FUNCTION_BLOCK FB_Syntax_Derived EXTENDS FB_Syntax_AbstractBase IMPLEMENTS I_Syntax_Extended
VAR
    _sStatus  : STRING := 'IDLE';
    _nCounter : DINT;
END_VAR

_nCounter := _nCounter + 1;

METHOD M_Execute : BOOL
VAR_INPUT
    nCommand : DINT;
END_VAR
CASE nCommand OF
    1:
        _sStatus := 'RUNNING';
    2:
        _sStatus := 'PAUSED';
ELSE
    _sStatus := 'UNKNOWN';
END_CASE
M_Execute := TRUE;
END_METHOD

METHOD M_GetValue : INT
M_GetValue := TO_INT(_nCounter);
END_METHOD

METHOD M_Reset : BOOL
_nCounter := 0;
_bReady   := TRUE;
_sStatus  := 'RESET';
M_Reset   := TRUE;
END_METHOD

PROPERTY P_ExtendedStatus : INT
GET
P_ExtendedStatus := 1;
END_GET
END_PROPERTY

PROPERTY P_Status : STRING
GET
P_Status := _sStatus;
END_GET
END_PROPERTY

END_FUNCTION_BLOCK

(* stored: Version 1.1.0.1, ProductVersion 3.1.4024.16
   POU FB_Syntax_Derived: Id {ee893be3-3f4d-43fd-ad98-be9638564c28}, SpecialFunc None
   Method M_Execute: Id {e5f6a1b2-c3d4-4e5f-c06b-7c8d9e0f1a2b}
   Method M_GetValue: Id {ab1b6ad1-a4ee-40bd-81ae-4c3f57901aec}
   Method M_Reset: Id {d4e5f6a1-b2c3-4d4e-bf5a-6b7c8d9e0f1a}
   Property P_ExtendedStatus: Id {acb160f8-190f-4161-806f-16a237f4e6af}
   Get Get: Id {5e573bf0-7431-42eb-99fa-2e7219b3fa95}
   Property P_Status: Id {f6a1b2c3-d4e5-4f6a-d17c-8d9e0f1a2b3c}
   Get Get: Id {a1b2c3d4-e5f6-4a7b-e28d-9e0f1a2b3c4d} *)
